{attribute 'GeneratedUsingTerminal: EK1100-0000-0018'}
{attribute addProperty BoxType "EK1100-0000-0018"}
{attribute addProperty Id "Beckhoff_EQ3xxxEK1122Beckhoff_EQ3xxxEK1122_66FBF7AB606"}
{attribute addProperty CRC "2939742606"}
{attribute addProperty Size "606"}
TYPE Beckhoff_EQ3xxx_AF38E98E EXTENDS EK1100_1FC0878B :
STRUCT
	{attribute addProperty Name "Beckhoff_EQ3xxxEK1122"}
	{attribute addProperty PreviousPort "Beckhoff EQ3xxx : B"}
	Beckhoff_EQ3xxxEK1122 : Beckhoff_EQ3xxxEK1122_66FBF7AB;
END_STRUCT
END_TYPE

(* stored: Version 1.2.0.0, ProductVersion 3.1.4024.9
   DUT Beckhoff_EQ3xxx_AF38E98E: Id {2d10ad49-b3bd-4d5f-9dfe-16ae28747938} *)
